// TIA Portal V15.1 export
// export: Created 2024-05-17T05:38:25.200442Z, ExportSetting WithDefaults, DisplayName Totally Integrated Automation Portal, DisplayVersion V15.1 Update 5, DisplayName TIA Portal Openness, DisplayVersion V15.1 Update 5, DisplayName SINAMICS Startdrive Advanced, DisplayVersion V15.1, DisplayName G130, G150, S120, S150, SINAMICS MV, S210, DisplayVersion V15.1, DisplayName G110M, G120, G120C, G120D, G120P, DisplayVersion V15.1, DisplayName STEP 7 Professional, DisplayVersion V15.1 Update 5, DisplayName STEP 7 Safety, DisplayVersion V15.1, DisplayName WinCC Professional, DisplayVersion V15.1 Update 5, DisplayName SIMATIC Visualization Architect, DisplayVersion V15.1
FUNCTION_BLOCK "LRedundantDet"   // FB1419, FBD
TITLE = LRedundantDet
{ S7_Optimized_Access := 'FALSE' }
AUTHOR : VCC
FAMILY : AlarmHnd
NAME : RedunDet
VERSION : 1.0
// ================================================================================
// This module is used everywhere 2 redundant detections are needed on working 
// area to avoid activation with safety shoes.
// If the alarm is enable, one alarm shall be generated
// when detection 1 is true and some time later the detection 2 is still false
// or when detection 2 is true and some time later the detection 1 is still false
// then Alarm is generated.
// Alarm is disable from HMI, a boolean output is available to inform the upper 
// level and do action in the Alarm summary.
// When the conditions to generate the alarm is disappear, a boolean output is 
// available to inform the upper level that the alarm can be reset.
// The alarm is reset by means of the AlarmResetPB signal.
// ================================================================================
// stored: AutoNumber false, IsIECCheckEnabled false, SetENOAutomatically False, UDAEnableTagReadback false
   VAR_INPUT
      I_Detection1 { ExternalAccessible := 'False'; ExternalVisible := 'False'; ExternalWritable := 'False'} : Bool;   // Input signal of detection 1
      I_Detection2 { ExternalAccessible := 'False'; ExternalVisible := 'False'; ExternalWritable := 'False'} : Bool;   // Input signal of detection 2
      I_EnableAlarm { ExternalAccessible := 'False'; ExternalVisible := 'False'; ExternalWritable := 'False'} : Bool := TRUE;   // Enable alarm from upper level
      I_Invisible { ExternalAccessible := 'False'; ExternalVisible := 'False'; ExternalWritable := 'False'} : Bool;   // Invisible
      I_AlarmResetPB { ExternalAccessible := 'False'; ExternalVisible := 'False'; ExternalWritable := 'False'} : Bool;   // Alarm reset pushbutton is activated
      I_TimeDelay { ExternalAccessible := 'False'; ExternalVisible := 'False'; ExternalWritable := 'False'} : DInt;   // Time delay value (1 unit = 1 ms)
      H_In : Struct   // HMI
         DisableAlarm : Bool;   // Disable alarm from HMI
      END_STRUCT;
   END_VAR
   VAR_OUTPUT
      O_RedundantDetAlm { ExternalAccessible := 'False'; ExternalVisible := 'False'; ExternalWritable := 'False'} : Bool;   // Redundant detection Alarm
      O_AlarmDisabled { ExternalAccessible := 'False'; ExternalVisible := 'False'; ExternalWritable := 'False'} : Bool;   // Alarm disabled from HMI
      O_AlarmABCondition { ExternalAccessible := 'False'; ExternalVisible := 'False'; ExternalWritable := 'False'} : Bool;   // Alarm AB condition
      H_IAnim { ExternalAccessible := 'False'; ExternalVisible := 'False'; ExternalWritable := 'False'} : Word;
      H_Out : Struct   // HMI
         Anim : Word;   // HMI Animation of the object
      END_STRUCT;
   END_VAR
   VAR DB_SPECIFIC
      DelayTimeResult { ExternalAccessible := 'False'; ExternalVisible := 'False'; ExternalWritable := 'False'} : Bool;   // Delay time boolean
      Detection1Mem { ExternalAccessible := 'False'; ExternalVisible := 'False'; ExternalWritable := 'False'} : Bool;   // Memory detyection 1 on true
      Detection2Mem { ExternalAccessible := 'False'; ExternalVisible := 'False'; ExternalWritable := 'False'} : Bool;   // Memory detyection 2 on true
      ResetDetectionMem { ExternalAccessible := 'False'; ExternalVisible := 'False'; ExternalWritable := 'False'} : Bool;   // condition to reset the detection memories
      SummaryRedundantDetAlm { ExternalAccessible := 'False'; ExternalVisible := 'False'; ExternalWritable := 'False'} : Bool;   // Summary redundant detection Alarm
      RedundantDetAlm { ExternalAccessible := 'False'; ExternalVisible := 'False'; ExternalWritable := 'False'} : Bool;   // Redundant detection Alarm
      RedundantDetAlmCond { ExternalAccessible := 'False'; ExternalVisible := 'False'; ExternalWritable := 'False'} : Bool;   // Redundant detection Alarm condition
   END_VAR
   VAR
      DelayTimer { ExternalAccessible := 'False'; ExternalVisible := 'False'; ExternalWritable := 'False'; S7_SetPoint := 'True'} : "LTimer";
   END_VAR
BEGIN

REGION Network 1: **** 2.2 - Alarms - Alarms Generation **** Creation of delay time
   // Creation of delay time
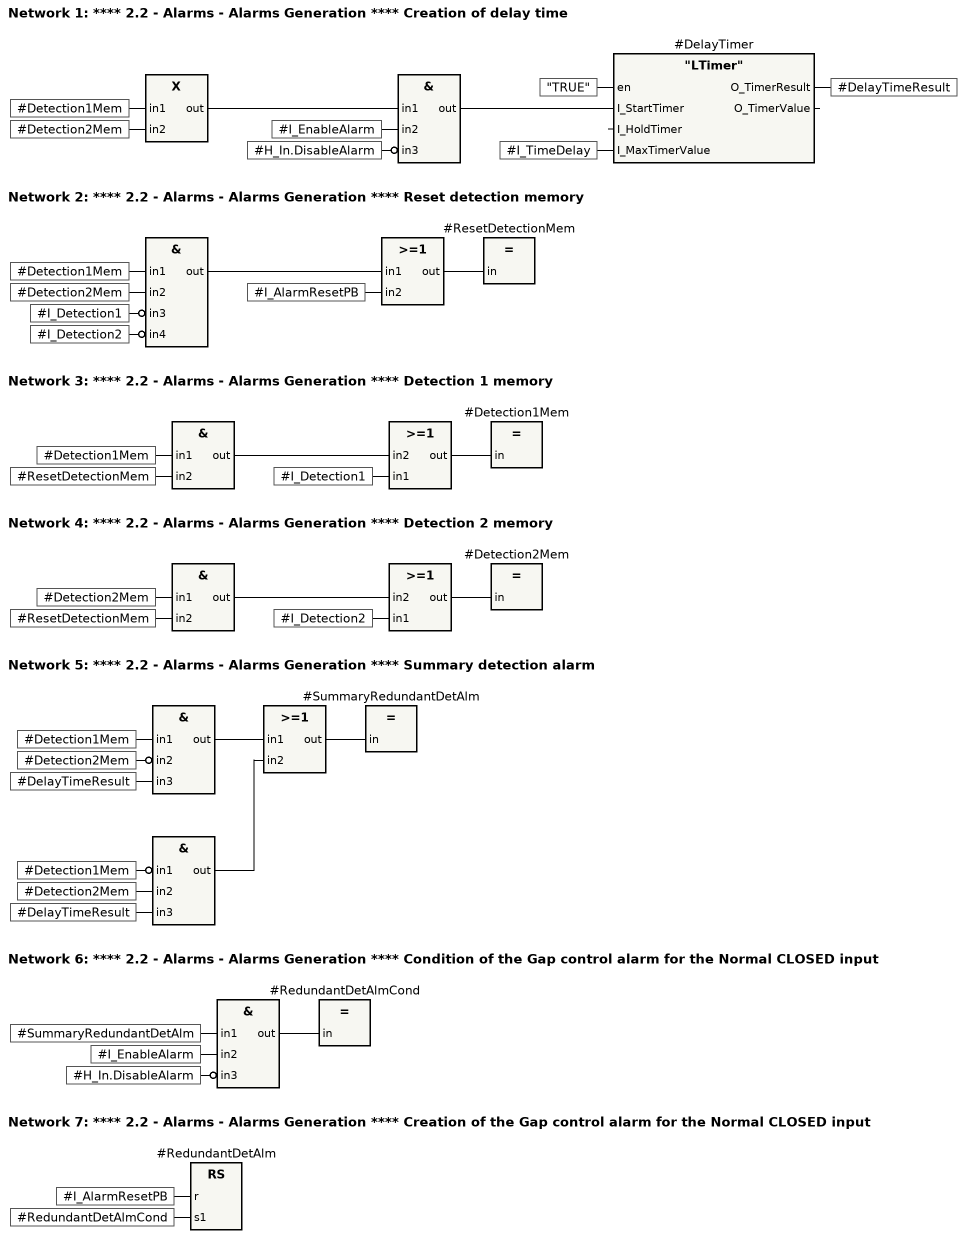
   IF "TRUE" THEN
       #DelayTimer(I_StartTimer := (#Detection1Mem XOR #Detection2Mem) AND #I_EnableAlarm AND NOT #H_In.DisableAlarm,   // "LTimer"
                   I_MaxTimerValue := #I_TimeDelay,
                   O_TimerResult => #DelayTimeResult);
   END_IF;
END_REGION

REGION Network 2: **** 2.2 - Alarms - Alarms Generation **** Reset detection memory
   // Reset detection memory
   #ResetDetectionMem := (#Detection1Mem AND #Detection2Mem AND NOT #I_Detection1 AND NOT #I_Detection2) OR #I_AlarmResetPB;
END_REGION

REGION Network 3: **** 2.2 - Alarms - Alarms Generation **** Detection 1 memory
   // Detection 1 memory
   #Detection1Mem := (#Detection1Mem AND #ResetDetectionMem) OR #I_Detection1;
END_REGION

REGION Network 4: **** 2.2 - Alarms - Alarms Generation **** Detection 2 memory
   // Detection 2 memory
   #Detection2Mem := (#Detection2Mem AND #ResetDetectionMem) OR #I_Detection2;
END_REGION

REGION Network 5: **** 2.2 - Alarms - Alarms Generation **** Summary detection alarm
   // Summary detection alarm
   #SummaryRedundantDetAlm := (#Detection1Mem AND NOT #Detection2Mem AND #DelayTimeResult) OR (NOT #Detection1Mem AND #Detection2Mem AND #DelayTimeResult);
END_REGION

REGION Network 6: **** 2.2 - Alarms - Alarms Generation **** Condition of the Gap control alarm for the Normal CLOSED input
   // Condition of the Gap control alarm for the Normal CLOSED input
   #RedundantDetAlmCond := #SummaryRedundantDetAlm AND #I_EnableAlarm AND NOT #H_In.DisableAlarm;
END_REGION

REGION Network 7: **** 2.2 - Alarms - Alarms Generation **** Creation of the Gap control alarm for the Normal CLOSED input
   // Creation of the Gap control alarm for the Normal CLOSED input
   IF #I_AlarmResetPB THEN
       #RedundantDetAlm := FALSE;   // RS flip-flop
   END_IF;
   IF #RedundantDetAlmCond THEN #RedundantDetAlm := TRUE; END_IF;
END_REGION

REGION Network 8: **** 4.6 - Mashine Status - Indications **** Icon Animation
   // Icon Animation
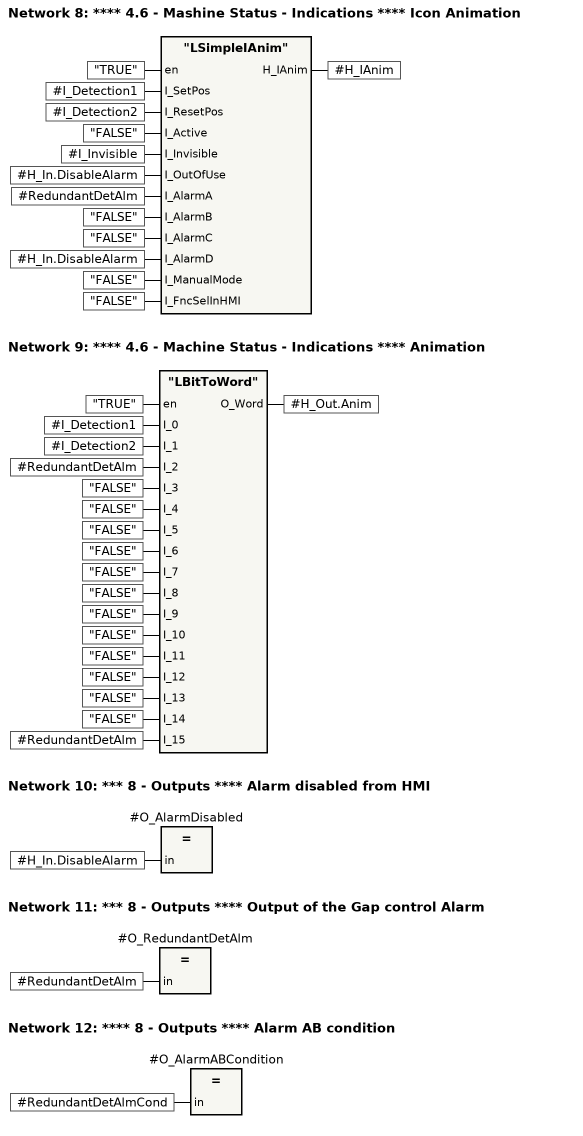
   IF "TRUE" THEN
       "LSimpleIAnim"(I_SetPos := #I_Detection1,
                      I_ResetPos := #I_Detection2,
                      I_Active := "FALSE",
                      I_Invisible := #I_Invisible,
                      I_OutOfUse := #H_In.DisableAlarm,
                      I_AlarmA := #RedundantDetAlm,
                      I_AlarmB := "FALSE",
                      I_AlarmC := "FALSE",
                      I_AlarmD := #H_In.DisableAlarm,
                      I_ManualMode := "FALSE",
                      I_FncSelInHMI := "FALSE",
                      H_IAnim => #H_IAnim);
   END_IF;
END_REGION

REGION Network 9: **** 4.6 - Machine Status - Indications **** Animation
   // Animation
   IF "TRUE" THEN
       "LBitToWord"(I_0 := #I_Detection1,
                    I_1 := #I_Detection2,
                    I_2 := #RedundantDetAlm,
                    I_3 := "FALSE",
                    I_4 := "FALSE",
                    I_5 := "FALSE",
                    I_6 := "FALSE",
                    I_7 := "FALSE",
                    I_8 := "FALSE",
                    I_9 := "FALSE",
                    I_10 := "FALSE",
                    I_11 := "FALSE",
                    I_12 := "FALSE",
                    I_13 := "FALSE",
                    I_14 := "FALSE",
                    I_15 := #RedundantDetAlm,
                    O_Word => #H_Out.Anim);
   END_IF;
END_REGION

REGION Network 10: *** 8 - Outputs **** Alarm disabled from HMI
   // Alarm disabled from HMI
   #O_AlarmDisabled := #H_In.DisableAlarm;
END_REGION

REGION Network 11: *** 8 - Outputs **** Output of the Gap control Alarm
   // Output of the Gap control Alarm
   #O_RedundantDetAlm := #RedundantDetAlm;
END_REGION

REGION Network 12: **** 8 - Outputs **** Alarm AB condition
   // Alarm AB condition
   #O_AlarmABCondition := #RedundantDetAlmCond;
END_REGION
END_FUNCTION_BLOCK
